// TIA Portal V16 export
// export: Created 2022-11-17T11:55:35.4326489Z, ExportSetting WithDefaults, DisplayName Totally Integrated Automation Portal, DisplayVersion V16 Update 6, DisplayName TIA Portal Version Control Interface, DisplayVersion V16 Update 2, DisplayName TIA Portal Openness, DisplayVersion V16 Update 6, DisplayName SINAMICS Startdrive Advanced, DisplayVersion V16 Update 5, DisplayName SINAMICS Startdrive G130, G150, S120, S150, SINAMICS MV, S210, DisplayVersion V16 Update 5, DisplayName SINAMICS Startdrive G110M, G120, G120C, G120D, G120P, G115D, DisplayVersion V16 Update 5, DisplayName STEP 7 Professional, DisplayVersion V16 Update 6, DisplayName STEP 7 Safety, DisplayVersion V16, DisplayName WinCC Advanced, DisplayVersion V16 Update 6
DATA_BLOCK "DB249_Program1"   // DB249
{ S7_Optimized_Access := 'FALSE' }
AUTHOR : Robopac
VERSION : 0.0
// stored: AutoNumber false, IsOnlyStoredInLoadMemory false, IsWriteProtectedInAS false
   VAR RETAIN
      Program1 { S7_SetPoint := 'True'} : "DatiProgramma";
   END_VAR
BEGIN
   Program1.Wrapping := TRUE;
   Program1.TopLenght := 500;
   Program1.TopRelease := 0;
   Program1.TopDown := 0;
   Program1.Top := 4;
   Program1.PressurePTime := 0;
   Program1.LifterTime := 0;
   Program1.RevOverContrast := 1;
   Program1.RopeEndCycle := 16#02;
   Program1.Spare4 := 16#01;
   Program1.RopeTime := 1500;
   Program1.RevOverClamp := 1;
   Program1.FilmForceFinalRev := 25;
   Program1.FilmPrestretchFinalRev := 100;
   Program1.ArmSpeed := 87;
   Program1.CarriageDown4Top := 500;
   Program1.TopDownTime := 1500;
   Program1.LapsUnderTop := 0;
   Program1.Spare6 := 0;
   Program1.Spare7 := 0;
   Program1.Spare8 := 0;
   Program1.Spare9 := 0;
   Program1.Spare10 := 0;
   Program1.Spare11 := 0;
   Program1.Spare12 := 0;
   Program1.Overlap0_1 := 0;
   Program1.Height1 := 120;
   Program1.Landmark1 := FALSE;
   Program1.Lifter1 := FALSE;
   Program1.SpareBit1H1 := FALSE;
   Program1.Airblower1 := TRUE;
   Program1.NextStep1 := TRUE;
   Program1.PressureP1 := TRUE;
   Program1.SpareByte2H1 := 16#00;
   Program1.Revolution1 := 1;
   Program1.RopeUnit1_1 := 16#03;
   Program1.RopeUnit1_2 := 16#01;
   Program1.FilmForce1 := 5;
   Program1.FilmPrestretch1 := 200;
   Program1.Spare3H1 := 0;
   Program1.Spare49 := 0;
   Program1.Spare50 := 0;
   Program1.Spare51 := 0;
   Program1.Spare52 := 0;
   Program1.Spare53 := 0;
   Program1.Overlap1_2 := 0;
   Program1.Height2 := 85;
   Program1.Landmark2 := FALSE;
   Program1.Lifter2 := FALSE;
   Program1.SpareBit1H2 := FALSE;
   Program1.Airblower2 := TRUE;
   Program1.NextStep2 := TRUE;
   Program1.PressureP2 := TRUE;
   Program1.SpareByte2H2 := 16#00;
   Program1.Revolution2 := 3;
   Program1.RopeUnit2_1 := 16#01;
   Program1.RopeUnit2_2 := 16#01;
   Program1.FilmForce2 := 15;
   Program1.FilmPrestretch2 := 200;
   Program1.Spare3H2 := 0;
   Program1.Spare54 := 0;
   Program1.Spare55 := 0;
   Program1.Spare56 := 0;
   Program1.Spare57 := 0;
   Program1.Spare58 := 0;
   Program1.Overlap2_3 := 300;
   Program1.Height3 := 110;
   Program1.Landmark3 := FALSE;
   Program1.Lifter3 := FALSE;
   Program1.SpareBit1H3 := FALSE;
   Program1.Airblower3 := TRUE;
   Program1.NextStep3 := TRUE;
   Program1.PressureP3 := TRUE;
   Program1.SpareByte2H3 := 16#00;
   Program1.Revolution3 := 2;
   Program1.RopeUnit3_1 := 16#03;
   Program1.RopeUnit3_2 := 16#03;
   Program1.FilmForce3 := 20;
   Program1.FilmPrestretch3 := 200;
   Program1.Spare3H3 := 0;
   Program1.Spare59 := 0;
   Program1.Spare60 := 0;
   Program1.Spare61 := 380;
   Program1.Spare62 := 2800;
   Program1.Spare63 := 0;
   Program1.Overlap3_4 := 100;
   Program1.Height4 := -100;
   Program1.Landmark4 := TRUE;
   Program1.Lifter4 := FALSE;
   Program1.SpareBit1H4 := FALSE;
   Program1.Airblower4 := FALSE;
   Program1.NextStep4 := TRUE;
   Program1.PressureP4 := TRUE;
   Program1.SpareByte2H4 := 16#00;
   Program1.Revolution4 := 1;
   Program1.RopeUnit4_1 := 16#01;
   Program1.RopeUnit4_2 := 16#01;
   Program1.FilmForce4 := 18;
   Program1.FilmPrestretch4 := 200;
   Program1.Spare3H4 := 0;
   Program1.Spare64 := 0;
   Program1.Spare65 := 0;
   Program1.Spare66 := 0;
   Program1.Spare67 := 0;
   Program1.Spare68 := 0;
   Program1.Overlap4_5 := 100;
   Program1.Height5 := 60;
   Program1.Landmark5 := FALSE;
   Program1.Lifter5 := FALSE;
   Program1.SpareBit1H5 := FALSE;
   Program1.Airblower5 := TRUE;
   Program1.NextStep5 := TRUE;
   Program1.PressureP5 := FALSE;
   Program1.SpareByte2H5 := 16#00;
   Program1.Revolution5 := 1;
   Program1.RopeUnit5_1 := 16#01;
   Program1.RopeUnit5_2 := 16#01;
   Program1.FilmForce5 := 25;
   Program1.FilmPrestretch5 := 200;
   Program1.Spare3H5 := 0;
   Program1.Spare69 := 0;
   Program1.Spare70 := 0;
   Program1.Spare71 := 0;
   Program1.Spare72 := 0;
   Program1.Spare73 := 0;
   Program1.Overlap5_6 := 100;
   Program1.Height6 := 40;
   Program1.Landmark6 := FALSE;
   Program1.Lifter6 := FALSE;
   Program1.SpareBit1H6 := FALSE;
   Program1.Airblower6 := TRUE;
   Program1.NextStep6 := FALSE;
   Program1.PressureP6 := FALSE;
   Program1.SpareByte2H6 := 16#00;
   Program1.Revolution6 := 1;
   Program1.RopeUnit6_1 := 16#01;
   Program1.RopeUnit6_2 := 16#01;
   Program1.FilmForce6 := 15;
   Program1.FilmPrestretch6 := 200;
   Program1.Spare3H6 := 0;
   Program1.Spare74 := 0;
   Program1.Spare75 := 0;
   Program1.Spare76 := 0;
   Program1.Spare77 := 0;
   Program1.Spare78 := 0;
   Program1.Overlap6_7 := 0;
   Program1.Height7 := 0;
   Program1.Landmark7 := FALSE;
   Program1.Lifter7 := FALSE;
   Program1.SpareBit1H7 := FALSE;
   Program1.Airblower7 := FALSE;
   Program1.NextStep7 := TRUE;
   Program1.PressureP7 := FALSE;
   Program1.SpareByte2H7 := 16#00;
   Program1.Revolution7 := 1;
   Program1.RopeUnit7_1 := 16#01;
   Program1.RopeUnit7_2 := 16#01;
   Program1.FilmForce7 := 0;
   Program1.FilmPrestretch7 := 100;
   Program1.Spare3H7 := 0;
   Program1.Spare79 := 0;
   Program1.Spare80 := 0;
   Program1.Spare81 := 0;
   Program1.Spare82 := 0;
   Program1.Spare83 := 0;
   Program1.Overlap7_8 := 0;
   Program1.Height8 := 0;
   Program1.Landmark8 := FALSE;
   Program1.Lifter8 := FALSE;
   Program1.SpareBit1H8 := FALSE;
   Program1.Airblower8 := FALSE;
   Program1.NextStep8 := TRUE;
   Program1.PressureP8 := FALSE;
   Program1.SpareByte2H8 := 16#00;
   Program1.Revolution8 := 1;
   Program1.RopeUnit8_1 := 16#01;
   Program1.RopeUnit8_2 := 16#01;
   Program1.FilmForce8 := 0;
   Program1.FilmPrestretch8 := 100;
   Program1.Spare3H8 := 0;
   Program1.Spare84 := 0;
   Program1.Spare85 := 0;
   Program1.Spare86 := 0;
   Program1.Spare87 := 0;
   Program1.Spare88 := 0;
   Program1.Overlap8_9 := 0;
   Program1.Height9 := 0;
   Program1.Landmark9 := FALSE;
   Program1.Lifter9 := FALSE;
   Program1.SpareBit1H9 := FALSE;
   Program1.Airblower9 := FALSE;
   Program1.NextStep9 := TRUE;
   Program1.PressureP9 := FALSE;
   Program1.SpareByte2H9 := 16#00;
   Program1.Revolution9 := 1;
   Program1.RopeUnit9_1 := 16#01;
   Program1.RopeUnit9_2 := 16#01;
   Program1.FilmForce9 := 0;
   Program1.FilmPrestretch9 := 100;
   Program1.Spare3H9 := 0;
   Program1.Spare89 := 0;
   Program1.Spare90 := 0;
   Program1.Spare91 := 0;
   Program1.Spare92 := 0;
   Program1.Spare93 := 0;
   Program1.Overlap9_10 := 0;
   Program1.Height10 := 0;
   Program1.Landmark10 := FALSE;
   Program1.Lifter10 := FALSE;
   Program1.SpareBit1H10 := FALSE;
   Program1.Airblower10 := FALSE;
   Program1.NextStep10 := FALSE;
   Program1.PressureP10 := FALSE;
   Program1.SpareByte2H10 := 16#00;
   Program1.Revolution10 := 1;
   Program1.RopeUnit10_1 := 16#01;
   Program1.RopeUnit10_2 := 16#01;
   Program1.FilmForce10 := 0;
   Program1.FilmPrestretch10 := 100;
   Program1.Spare3H10 := 0;
   Program1.Spare94 := 0;
   Program1.Spare95 := 0;
   Program1.Spare96 := 0;
   Program1.Spare97 := 0;
   Program1.Spare98 := 0;
   Program1.Overlap10_11 := 0;
   Program1.Height11 := 0;
   Program1.Landmark11 := FALSE;
   Program1.Lifter11 := FALSE;
   Program1.SpareBit1H11 := FALSE;
   Program1.Airblower11 := FALSE;
   Program1.NextStep11 := TRUE;
   Program1.PressureP11 := FALSE;
   Program1.SpareByte2H11 := 16#00;
   Program1.Revolution11 := 1;
   Program1.RopeUnit11_1 := 16#01;
   Program1.RopeUnit11_2 := 16#01;
   Program1.FilmForce11 := 0;
   Program1.FilmPrestretch11 := 100;
   Program1.Spare3H11 := 0;
   Program1.Spare99 := 0;
   Program1.Spare100 := 0;
   Program1.Spare101 := 0;
   Program1.Spare102 := 0;
   Program1.Spare103 := 0;
   Program1.Overlap11_12 := 0;
   Program1.Height12 := 0;
   Program1.Landmark12 := FALSE;
   Program1.Lifter12 := FALSE;
   Program1.SpareBit1H12 := FALSE;
   Program1.Airblower12 := FALSE;
   Program1.NextStep12 := FALSE;
   Program1.PressureP12 := FALSE;
   Program1.SpareByte2H12 := 16#00;
   Program1.Revolution12 := 1;
   Program1.RopeUnit12_1 := 16#01;
   Program1.RopeUnit12_2 := 16#01;
   Program1.FilmForce12 := 0;
   Program1.FilmPrestretch12 := 100;
   Program1.Spare3H12 := 0;
   Program1.Spare104 := 0;
   Program1.Spare105 := 0;
   Program1.Spare106 := 0;
   Program1.Spare107 := 0;
   Program1.Spare108 := 0;
END_DATA_BLOCK
